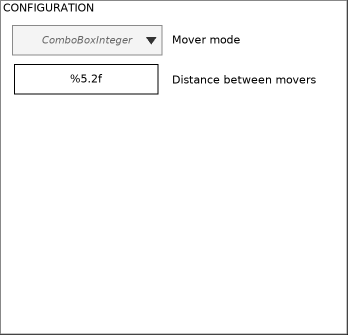
VISUALIZATION VI_XTSConfigurationVisu  // 348x335
VAR_IN_OUT
	xts : XTS_System;
END_VAR
    Rectangle (0,0 348x335), "CONFIGURATION"
    Label (169,25 150x30), "Mover mode"
    ComboBoxInteger (12,25 150x30), variable: xts.stCfg.udiMoverMode, text list: 'MoverMode_TXT'
    Label (169,65 150x30), "Distance between movers"
    Rectangle (14,64 144x30), "%5.2f", text variable: xts.stCfg.lrMoverDistance
        OnMouseClick: write the text variable via Default
END_VISUALIZATION

(* stored: Version 1.1.0.1, ProductVersion 3.1.4024.11
   Visu VI_XTSConfigurationVisu: Id {063e2089-6a55-47b1-b0c7-c8644bd955c4} *)
